Fanuc KAREL source: kf00104.KL

-- PROVISIONAL review KL for V770-1; original PC SHA256 f84e24be7311fffb1172d37c478ef2111357ea72d326254ee18451900b1304ae
-- Incomplete behavior may be omitted. Consult companion uncertainty JSON. Do not deploy.
PROGRAM KF00104
%NOLOCKGROUP
BEGIN
  -- UNRESOLVED_PC offsets 5-16; opcodes 2E,23
  -- UNRESOLVED_PC offsets 21-32; opcodes 2E,23
  -- UNRESOLVED_PC offsets 37-57; opcodes 27,27,9D,22,2A,22,31
  -- UNRESOLVED_PC offsets 62-66; opcodes 7F
END KF00104
